FUNCTION_BLOCK FB_Cylinder_DualSolenoid_DualSensor EXTENDS FB_Cylinder_DualSensor
VAR_INPUT
END_VAR
VAR_OUTPUT
END_VAR
VAR
	bExtend_Actuator_HardwareOutput 	AT %Q* 	: BOOL;
	bRetract_Actuator_HardwareOutput 	AT %Q* 	: BOOL;
END_VAR

METHOD HardwareUpdate : BOOL
VAR_INPUT
END_VAR
SUPER^.HardwareUpdate();

bExtend_Actuator_HardwareOutput := bExtendCommand;
bRetract_Actuator_HardwareOutput := bRetractCommand;
END_METHOD

END_FUNCTION_BLOCK

(* stored: Version 1.1.0.1, ProductVersion 3.1.4024.9
   POU FB_Cylinder_DualSolenoid_DualSensor: Id {54913be8-2f9a-4c62-91f9-7183be15cd2e}, SpecialFunc None
   Folder 01_SUPER_Overrides: Id {b1091b7f-7b7c-40ae-923e-78fa7db5ad15}
   Method HardwareUpdate: Id {1a62f8fc-8df7-4ab8-a437-e384e4ffc47d} *)
